// TIA Portal V18 export
DATA_BLOCK "deleter"   // DB66
VERSION : 0.1
// stored: AutoNumber true, DBAccessibleFromOPCUA true, InstanceOfName _ML2_ts_block1, InstanceOfType FB
"_ML2_ts_block1"
   // VAR_INPUT
   //    R_ALL : Bool;
   //    SwAuto : Bool;
   //    AutoRuning : Bool;
   //    Arrived : Bool;
   //    R_SeimAuto : Bool;
   //    CLK_Spot : Bool;
   //    CLK_Defect : Bool;
   //    CLK_Home : Bool;
   //    CLK_Load : Bool;
   //    CLK_Control2 : Bool;
   //    CLK_Control1 : Bool;
   // END_VAR
   // VAR_OUTPUT
   //    Q0_Auto : Bool;
   //    q0_AutoWaiting : Bool;
   //    Q0_SemiAuto : Bool;
   //    P1_Spot : Bool;
   //    Q1_Spot : Bool;
   //    P2_Defect : Bool;
   //    Q2_Defect : Bool;
   //    P3_Home : Bool;
   //    Q3_Home : Bool;
   //    P4_Load : Bool;
   //    Q4_Load : Bool;
   //    P5_Control1 : Bool;
   //    Q5_Control1 : Bool;
   //    P6_Control2 : Bool;
   //    Q6_control2 : Bool;
   //    Q99_none : Bool;
   //    Q99_Any : Bool;
   // END_VAR
   // VAR
   //    memarrived : Bool;
   //    reset_Qs : Bool;
   //    last_button_stands_Instance { S7_SetPoint := 'True'} : "last_button_stands";
   //    Q_integer { S7_SetPoint := 'True'} : Int;
   //    trDefect { S7_SetPoint := 'True'} : R_TRIG;
   //    trSpot { S7_SetPoint := 'True'} : R_TRIG;
   //    bsu_Spot { S7_SetPoint := 'True'} : "_ML2_ts_block1_subunit";
   //    bsu_Defect { S7_SetPoint := 'True'} : "_ML2_ts_block1_subunit";
   //    bsuHome { S7_SetPoint := 'True'} : "_ML2_ts_block1_subunit";
   //    bsu_load { S7_SetPoint := 'True'} : "_ML2_ts_block1_subunit";
   //    bsuControl1 { S7_SetPoint := 'True'} : "_ML2_ts_block1_subunit";
   //    bsuControl2 { S7_SetPoint := 'True'} : "_ML2_ts_block1_subunit";
   // END_VAR
BEGIN
END_DATA_BLOCK
